VAR_GLOBAL
	Button_Open : BOOL;
	Button_Close : BOOL;
	Sensor_Open : BOOL;
	Sensor_Close : BOOL;
	System_Status : STRING := 'READY';
	Motor_Moving : BOOL;
	Light_Output : BOOL;
	Safety_Sensor :BOOL;
	
END_VAR

(* stored: Version 1.1.0.1, ProductVersion 3.1.4024.15
   GVL Variables: Id {a9a6ec33-2a75-406e-b38a-ade54feabb95} *)
